(* PLC project TC3_TE1400_GeneratedModule_TctSmplTempCtrl__FB, Beckhoff Automation GmbH & Co. KG TwinCAT 3 Function - TE1400 1.2.1230 *)
(* stored: companyURL www.beckhoff.com, creationDateTime 2018-02-26T08:09:58 *)

TYPE E_TcMatSimDataAreaType : (NotSpecified := 0, Standard, InputSrc, InputDst, OutputSrc, OutputDst, InternalDa, MArea, RetainDa);
END_TYPE

TYPE ST_TcMatSimObjectDataAreaInfo : STRUCT
  pPlcVar : PVOID;
  pModuleProcImg : PVOID;
  nSize : UDINT;
  nDataAreaId : UDINT;
  eDataAreaType : E_TcMatSimDataAreaType;
END_STRUCT;
END_TYPE

{attribute 'pack_mode' := '4'}
TYPE ST_TctSmplTempCtrl_InitData : STRUCT
  Header : TComInitDataHdr;
  CallByHdr : TComInitDataElmHdr;
  CallBy : TctModuleCallByType;
  ExecutionSequenceHdr : TComInitDataElmHdr;
  ExecutionSequence : TctModuleExecutionSequenceType;
  StepSizeHdr : TComInitDataElmHdr;
  StepSize : TctStepSizeType;
  ExtModeParametersHdr : TComInitDataElmHdr;
  ExtModeParameters : TctExtModeParametersType;
  ExecuteModelCodeHdr : TComInitDataElmHdr;
  ExecuteModelCode : BOOL;
  ModelParametersHdr : TComInitDataElmHdr;
  ModelParameters : P_TctSmplTempCtrl_T;
  ContextInfoArr_0_TaskOidHdr : TComInitDataElmHdr;
  ContextInfoArr_0_TaskOid : OTCID;
  ContextInfoArr_0_TaskPriorityHdr : TComInitDataElmHdr;
  ContextInfoArr_0_TaskPriority : UDINT;
  ContextInfoArr_0_TaskCycleTimeNsHdr : TComInitDataElmHdr;
  ContextInfoArr_0_TaskCycleTimeNs : UDINT;
  ContextInfoArr_0_TaskPortHdr : TComInitDataElmHdr;
  ContextInfoArr_0_TaskPort : UINT;
  ContextInfoArr_0_TaskSortOrderHdr : TComInitDataElmHdr;
  ContextInfoArr_0_TaskSortOrder : UDINT;
END_STRUCT;
END_TYPE

TYPE ST_TctSmplTempCtrl_Input : STRUCT
  FeedbackTemp : INT;
END_STRUCT;
END_TYPE

TYPE ST_TctSmplTempCtrl_Output : STRUCT
  HeaterOn : BOOL;
  MonitoringSignals : MonitoringSignalsType;
END_STRUCT;
END_TYPE

FUNCTION_BLOCK FB_TcMatSimObject
  VAR_INPUT
    bWriteFbInputValues : BOOL := TRUE;  (* set this flag to write FB input values to the TcComObject's input DataAreas. This will overwrite the mapped input values before module execution. Set to FALSE to read the mapped input values from the TcComObject to the FB. *)
  END_VAR
  VAR
    pDataAreas : POINTER TO ST_TcMatSimObjectDataAreaInfo;  (* process image src and dst pointers and sizes *)
    nDataAreas : UDINT;
    ipObjSrv : ITComObjectServer;  (* global interface pointers *)
    ipTcComObj : ITComObject;  (* object interface pointers *)
    ipTcCyclic : ITcCyclic;
    ipTcPostCyclic : ITcPostCyclic;
    ipTcAdi : ITcADI;
    ipTask : ITcTask;  (* task interface pointers *)
    pInitData : POINTER TO TComInitDataHdr;  (* initial parameters *)
    hResult : HRESULT;  (* hResult of interface calls (0 if no error) *)
    moduleClsId : CLSID;  (* module class ID *)
    assignedClsId : CLSID;  (* expected/desired module class ID *)
    bClassIdVerified : BOOL;
    bDynInstance : BOOL;  (* flag indicating whether the module instance was created dynamically *)
    eInitialObjState : TCOM_STATE := TCOM_STATE.TCOM_STATE_INIT;  (* the object state at the time FB_init was called, FB_exit will try to switch to this state (only if this means to shift down) *)
  END_VAR

            
          

{attribute 'object_name' := 'ReleaseTcComInterface'}
METHOD ReleaseTcComInterface : HRESULT
  VAR
    nStateChangeCnt : DINT := 0;
  END_VAR
                  
IF (ipTcComObj<>0) THEN
  WHILE (State>eInitialObjState AND nStateChangeCnt<1000) DO
    State := eInitialObjState;
    nStateChangeCnt := nStateChangeCnt+1;
  END_WHILE
  ReleaseObjInterfaces();
  IF (bDynInstance) THEN
    ReleaseTcComInterface := TC3_MODULE.FW_ObjMgr_DeleteInstance(ADR(ipTcComObj));
  ELSE
    ipTcComObj.TcRelease();
  END_IF
  ipTcComObj := 0;
END_IF
                  
                
END_METHOD

{attribute 'object_name' := 'ReleaseObjInterfaces'}
METHOD ReleaseObjInterfaces : HRESULT
                  
// release interface pointers
IF (ipTcCyclic<>0) THEN
  ipTcCyclic.TcRelease();
  ipTcCyclic := 0;
END_IF
IF (ipTcPostCyclic<>0) THEN
  ipTcPostCyclic.TcRelease();
  ipTcPostCyclic := 0;
END_IF
IF (ipTcAdi<>0) THEN
  ipTcAdi.TcRelease();
  ipTcAdi := 0;
END_IF
                  
                
END_METHOD

{attribute 'object_name' := 'Internal_SetObjState'}
METHOD Internal_SetObjState
  VAR_INPUT
    hr : REFERENCE TO HRESULT;
    nextState : TCOM_STATE;
  END_VAR
                  
// verify class id
IF (SUCCEEDED(hr)) THEN
  hr := VerifyClassId();
END_IF

// switch object state
IF (SUCCEEDED(hr) AND nextState>=TCOM_STATE_INIT) THEN
  IF (ipTcComObj=0) THEN
    hr := Tc2_System.E_HRESULTAdsErr.NOINTERFACE;
  END_IF
  IF (ipObjSrv=0) THEN
    hr := Tc2_System.E_HRESULTAdsErr.NOINTERFACE;
  END_IF
  IF (SUCCEEDED(hr)) THEN
    hr := ipTcComObj.TcSetObjState(nextState,ipObjSrv,pInitData);
  END_IF
END_IF
                  
                
END_METHOD

{attribute 'object_name' := 'FB_init'}
METHOD FB_init : BOOL
  VAR_INPUT
    bInitRetains : BOOL;  (* init retain variables *)
    bInCopyCode : BOOL;  (* Online Change *)
    oid : OTCID;
  END_VAR
                  
FB_init := SUCCEEDED(Init(oid));
                  
                
END_METHOD

{attribute 'object_name' := 'GetObjPara'}
METHOD GetObjPara : HRESULT
  VAR_INPUT
    pid : PTCID;
    nData : UDINT;
    pData : PVOID;
  END_VAR
                  
IF (ipTcComObj=0) THEN
  GetObjPara := Tc2_System.E_HRESULTAdsErr.NOINTERFACE;
END_IF

IF (SUCCEEDED(GetObjPara)) THEN
  GetObjPara := ipTcComObj.TcGetObjPara(pid:=pid,nData,pData,0);
END_IF
                  
                
END_METHOD

{attribute 'object_name' := 'QueryObjInterface'}
METHOD QueryObjInterface
  VAR_INPUT
    hr : REFERENCE TO HRESULT;
    iid : REFERENCE TO IID;
    pipItf : POINTER TO ITcUnknown;
  END_VAR
  VAR CONSTANT
    pNull : PVOID := 0;
  END_VAR
                  
IF (SUCCEEDED(hr)) THEN
  IF (ipTcComObj=0) THEN
    hr := Tc2_System.E_HRESULTAdsErr.NOINTERFACE;
  ELSIF (pipItf^=ULINT_TO_DWORD(pNull)) THEN
    hr := ipTcComObj.TcQueryInterface(iid:= iid, pipItf:=pipItf);
  END_IF
END_IF
                  
                
END_METHOD

{attribute 'object_name' := 'SaveOnlineParametersForInit'}
METHOD SaveOnlineParametersForInit : HRESULT
  VAR
    idx : UINT;
    pInitElemHdr : POINTER TO TComInitDataElmHdr;
    pData : PVOID;
    nData : UDINT;
  END_VAR
  VAR CONSTANT
    nInitDataAlignment : UDINT := 4;
  END_VAR
                  IF (pInitData<>0) THEN
  pInitElemHdr := pInitData + SIZEOF(pInitData^);
  FOR idx:=1 TO pInitData^.uiElmCnt DO
    pData := pInitElemHdr + ULINT_TO_DWORD(SIZEOF(pInitElemHdr^));
    nData := pInitElemHdr^.cbData;
    SaveOnlineParametersForInit := GetObjPara(pInitElemHdr^.indexOffset,nData,pData);
    IF (FAILED(SaveOnlineParametersForInit)) THEN
      RETURN;
    END_IF
    pInitElemHdr := pData + (nInitDataAlignment*((nData + nInitDataAlignment - 1)/nInitDataAlignment));
  END_FOR
ELSE
	SaveOnlineParametersForInit := Tc2_System.E_HRESULTAdsErr.NOTINIT;
END_IF
                  
                
END_METHOD

{attribute 'object_name' := 'ResetHresult'}
METHOD ResetHresult
                  hResult := S_OK;
                
END_METHOD

{attribute 'object_name' := 'Execute'}
METHOD Execute : HRESULT
  VAR
    nDaIdx : UDINT;
    pCurDataArea : POINTER TO ST_TcMatSimObjectDataAreaInfo;
  END_VAR
                  
IF (SUCCEEDED(hResult)) THEN
  hResult := VerifyClassId();
END_IF

IF (SUCCEEDED(hResult) AND State<>TCOM_STATE_OP) THEN
  hResult := Tc2_System.E_HRESULTAdsErr.NOTREADY;
END_IF

// get image pointers
IF (SUCCEEDED(hResult)) THEN
  GetImagePtrs(hResult);
END_IF

// copy inputs
IF (pDataAreas<>0 AND nDataAreas>0 AND bWriteFbInputValues) THEN
  FOR nDaIdx:=0 TO nDataAreas-1 DO
    IF (FAILED(hResult))THEN
      CONTINUE;
    END_IF
    pCurDataArea := pDataAreas + nDaIdx*SIZEOF(ST_TcMatSimObjectDataAreaInfo);
    IF ((pCurDataArea^.eDataAreaType <> E_TcMatSimDataAreaType.InputDst))THEN
      CONTINUE;
    END_IF
    IF (pCurDataArea^.pModuleProcImg<>0 AND pCurDataArea^.pPlcVar<>0) THEN
      MEMCPY(pCurDataArea^.pModuleProcImg,pCurDataArea^.pPlcVar,pCurDataArea^.nSize);
    ELSE
      hResult := Tc2_System.E_HRESULTAdsErr.NOINTERFACE;
    END_IF
  END_FOR
END_IF

// call cycle update
IF (SUCCEEDED(hResult)) THEN
  IF (ipTcCyclic<>0) THEN
    hResult := ipTcCyclic.CycleUpdate(ipTask:= ipTask, ipCaller:= 0, context:= 0);
  ELSE
    hResult := Tc2_System.E_HRESULTAdsErr.NOINTERFACE;
  END_IF
END_IF

// copy outputs
IF (pDataAreas<>0 AND nDataAreas>0) THEN
  FOR nDaIdx:=0 TO nDataAreas-1 DO
    IF (FAILED(hResult))THEN
      CONTINUE;
    END_IF
    pCurDataArea := pDataAreas + nDaIdx*SIZEOF(ST_TcMatSimObjectDataAreaInfo);
    IF ((pCurDataArea^.eDataAreaType = E_TcMatSimDataAreaType.OutputSrc) OR NOT bWriteFbInputValues) THEN
      IF (pCurDataArea^.pModuleProcImg<>0 AND pCurDataArea^.pPlcVar<>0) THEN
        MEMCPY(pCurDataArea^.pPlcVar,pCurDataArea^.pModuleProcImg,pCurDataArea^.nSize);
      ELSE
        hResult := Tc2_System.E_HRESULTAdsErr.NOINTERFACE;
      END_IF
    END_IF
  END_FOR
END_IF


// call post cyclic update
IF (SUCCEEDED(hResult)) THEN
  IF (ipTcPostCyclic<>0) THEN
    hResult := ipTcPostCyclic.PostCyclicUpdate(ipTask:= 0, ipCaller:= 0, context:= 0);
  ELSE
    hResult := Tc2_System.E_HRESULTAdsErr.NOINTERFACE;
  END_IF
END_IF

ReleaseImagePtrs();

Execute := hResult;
                  
                
END_METHOD

{attribute 'object_name' := 'GetImagePtrs'}
METHOD GetImagePtrs
  VAR_INPUT
    hr : REFERENCE TO HRESULT;
  END_VAR
  VAR
    nDaIdx : UDINT;
    pCurDataArea : POINTER TO ST_TcMatSimObjectDataAreaInfo;
  END_VAR
                  
IF (ipTcAdi=0) THEN
  hr := Tc2_System.E_HRESULTAdsErr.NOINTERFACE;
END_IF
IF(State<>TCOM_STATE_OP)THEN
  hr := Tc2_System.E_HRESULTAdsErr.INVALIDSTATE;
END_IF


// get pointers to process images
IF (pDataAreas<>0 AND nDataAreas>0) THEN
  FOR nDaIdx:=0 TO nDataAreas-1 DO
    pCurDataArea := pDataAreas + nDaIdx*SIZEOF(ST_TcMatSimObjectDataAreaInfo);
    IF (FAILED(hr))THEN
      CONTINUE;
    END_IF
    IF ((pCurDataArea^.eDataAreaType <> E_TcMatSimDataAreaType.InputDst) AND (pCurDataArea^.eDataAreaType <> E_TcMatSimDataAreaType.OutputSrc))THEN
      CONTINUE;
    END_IF
    IF (pCurDataArea^.pModuleProcImg=0 AND pCurDataArea^.nSize>0) THEN
      hr := ipTcAdi.GetImagePtr(size:= pCurDataArea^.nSize , offs:=0 , adi_x:=pCurDataArea^.nDataAreaId , ppData:=ADR(pCurDataArea^.pModuleProcImg));
    END_IF
  END_FOR
END_IF

IF (FAILED(hr)) THEN
  ReleaseImagePtrs();
END_IF
                  
                
END_METHOD

{attribute 'object_name' := 'VerifyClassId'}
METHOD VerifyClassId : HRESULT
  VAR
    emptyClsId : CLSID;
  END_VAR
                  memset(ADR(emptyClsId),0,SIZEOF(emptyClsId));
IF (bClassIdVerified) THEN
  // class ID was already verified
  VerifyClassId := Tc2_System.E_HRESULTAdsErr.HRESULT_ADS_NOERROR;
ELSIF (memcmp(ADR(assignedClsId),ADR(emptyClsId),SIZEOF(assignedClsId))=0) THEN
  // skip class ID verification if no assignedClsId specified
  VerifyClassId := Tc2_System.E_HRESULTAdsErr.HRESULT_ADS_NOERROR;
ELSE
  // verify class ID
  VerifyClassId := ReadModuleClassId();

  IF (SUCCEEDED(VerifyClassId)) THEN
    IF (memcmp(ADR(assignedClsId),ADR(moduleClsId),SIZEOF(assignedClsId))<>0) THEN
     VerifyClassId := Tc2_System.E_HRESULTAdsErr.INVALIDCLSID;
    END_IF
  END_IF
  bClassIdVerified := SUCCEEDED(VerifyClassId);
END_IF
                  
                
END_METHOD

{attribute 'object_name' := 'SetObjPara'}
METHOD SetObjPara : HRESULT
  VAR_INPUT
    pid : PTCID;
    nData : UDINT;
    pData : PVOID;
  END_VAR
                  
IF (ipTcComObj=0) THEN
  SetObjPara := Tc2_System.E_HRESULTAdsErr.NOINTERFACE;
END_IF

IF (SUCCEEDED(SetObjPara)) THEN
  SetObjPara := ipTcComObj.TcSetObjPara(pid:=pid,nData,pData,0);
END_IF
                  
                
END_METHOD

{attribute 'object_name' := 'QueryTcComInterface'}
METHOD QueryTcComInterface
  VAR_INPUT
    hr : REFERENCE TO HRESULT;
    oid : OTCID;
  END_VAR
                  
IF (ipObjSrv=0) THEN
  hr := Tc2_System.E_HRESULTAdsErr.NOINTERFACE;
END_IF

IF (SUCCEEDED(hr) AND ipTcComObj=0) THEN
  bDynInstance := FALSE;
  IF(oid>0) THEN
    // query interface of existing object
    hr := ipObjSrv.TcQueryObjectInterface(oid,IID_ITComObject,ADR(ipTcComObj));
  ELSE
    // create new instance and get the object interface
    hr := ipObjSrv.TcCreateInstance(assignedClsId,IID_ITComObject,ADR(ipTcComObj));
    IF (SUCCEEDED(hr)) THEN
      bDynInstance := TRUE;
      hr := ipTcComObj.TcSetObjectId(OTCID_CreateNewId);
    END_IF
  END_IF
  IF (SUCCEEDED(hr)) THEN
    eInitialObjState := State;
  END_IF
END_IF
                  
                
END_METHOD

{attribute 'object_name' := 'ReleaseImagePtrs'}
METHOD ReleaseImagePtrs : HRESULT
  VAR
    nDaIdx : UDINT;
    pCurDataArea : POINTER TO ST_TcMatSimObjectDataAreaInfo;
  END_VAR
                  
IF (ipTcAdi=0) THEN
  ReleaseImagePtrs := Tc2_System.E_HRESULTAdsErr.NOINTERFACE;
END_IF

IF (SUCCEEDED(ReleaseImagePtrs) AND pDataAreas<>0 AND nDataAreas>0) THEN
  // release pointers to the simulink module process images
  FOR nDaIdx:=0 TO nDataAreas-1 DO
    pCurDataArea := pDataAreas + nDaIdx*SIZEOF(ST_TcMatSimObjectDataAreaInfo);

    IF (pCurDataArea^.pModuleProcImg<>0) THEN
      ipTcAdi.ReleaseImagePtr(pData:=pCurDataArea^.pModuleProcImg);
      pCurDataArea^.pModuleProcImg := 0;
    END_IF
  END_FOR
END_IF
                  
                
END_METHOD

{attribute 'object_name' := 'FB_exit'}
METHOD FB_exit : BOOL
  VAR_INPUT
    bInCopyCode : BOOL;  (* Online Change *)
  END_VAR
                  
IF (NOT bInCopyCode) THEN
  IF (ipObjSrv<>0) THEN
    ipObjSrv.TcRelease();
    ipObjSrv := 0;
  END_IF

  ReleaseTcComInterface();
END_IF
                  
                
END_METHOD

{attribute 'object_name' := 'InitObjName'}
METHOD InitObjName
  VAR_INPUT
    hr : REFERENCE TO HRESULT;
  END_VAR
  VAR
    objectName : STRING(255) := 'TcMatSimObject_PlcRtFbInstance';
    oid : OTCID;
  END_VAR
                  
IF (SUCCEEDED(hr)) THEN
  hr := ipTcComObj.TcGetObjectId(oid);
END_IF

IF (SUCCEEDED(hr) and bDynInstance) THEN
  objectName := TC2_STANDARD.CONCAT(objectName,'_');
  objectName := TC2_STANDARD.CONCAT(objectName,UDINT_TO_STRING(oid));
  hr := ipTcComObj.TcSetObjectName(ADR(objectName));
END_IF
                  
                
END_METHOD

{attribute 'object_name' := 'SetObjState'}
METHOD SetObjState : HRESULT
  VAR_INPUT
    finalState : TCOM_STATE;
  END_VAR
  VAR
    bShiftUp : BOOL;
    bShiftDown : BOOL;
    currentState : TCOM_STATE;
  END_VAR
                  
currentState := State;

bShiftUp := finalState>currentState;
bShiftDown := finalState<currentState;

// do not switch up on error
IF (FAILED(hresult)) THEN
  bShiftUp := FALSE;
END_IF
// reset existing error on switching down
IF (bShiftDown) THEN
  ResetHresult();
END_IF

// prepared state switch
CASE currentState OF
  TCOM_STATE_INIT:
    IF(bShiftUp) THEN
      QueryTcComInterface(hResult,0);
      Internal_SetObjState(hResult,TCOM_STATE.TCOM_STATE_PREOP);
      InitObjName(hResult);
    END_IF

  TCOM_STATE_PREOP:
    IF(bShiftUp) THEN
      Internal_SetObjState(hResult,TCOM_STATE.TCOM_STATE_SAFEOP);
      QueryObjInterfaces(hResult);
    ELSIF (bShiftDown) THEN
      Internal_SetObjState(hResult,TCOM_STATE.TCOM_STATE_INIT);
    END_IF

  TCOM_STATE_SAFEOP:
    IF(bShiftUp) THEN
      Internal_SetObjState(hResult,TCOM_STATE.TCOM_STATE_OP);
      QueryObjInterfaces(hResult);
    ELSIF (bShiftDown) THEN
      Internal_SetObjState(hResult,TCOM_STATE.TCOM_STATE_PREOP);
      ReleaseObjInterfaces();
    END_IF


  TCOM_STATE_OP:
    IF (bShiftDown) THEN
      Internal_SetObjState(hResult,TCOM_STATE.TCOM_STATE_SAFEOP);
    END_IF
END_CASE

SetObjState := hResult;
                  
                
END_METHOD

{attribute 'object_name' := 'QueryObjInterfaces'}
METHOD QueryObjInterfaces
  VAR_INPUT
    hr : REFERENCE TO HRESULT;
  END_VAR
                  
IF(State<TCOM_STATE_PREOP)THEN
  hr := Tc2_System.E_HRESULTAdsErr.INVALIDSTATE;
END_IF

//cyclic interface
QueryObjInterface(hr,IID_ITCCYCLIC,ADR(ipTcCyclic));
//post cyclic interface
QueryObjInterface(hr,IID_ITCPOSTCYCLIC,ADR(ipTcPostCyclic));
//adi interface
QueryObjInterface(hr,IID_ITcADI,ADR(ipTcAdi));
                  
                
END_METHOD

{attribute 'object_name' := 'Init'}
METHOD Init : HRESULT
  VAR_INPUT
    oid : OTCID;
  END_VAR
                  
// preinitialize variables
memset(ADR(moduleClsId),0,SIZEOF(moduleClsId));
bClassIdVerified := FALSE;
hResult := Tc2_System.E_HRESULTAdsErr.HRESULT_ADS_NOERROR;

// get object server
IF (ipObjSrv=0) THEN
  hResult := FW_ObjMgr_GetObjectServer(_AppInfo.ObjId,ADR(ipObjSrv));
END_IF

// try to get object interfaces
IF (SUCCEEDED(hresult)) THEN
  QueryTcComInterface(hResult,oid);
END_IF

// verify class id
IF (SUCCEEDED(hresult)) THEN
  hresult := VerifyClassId();
END_IF

// query interfaces, if the current state is higher than INIT
IF (SUCCEEDED(hresult) AND State>TCOM_STATE.TCOM_STATE_INIT) THEN
  QueryObjInterfaces(hResult);
END_IF

// return value
Init := hresult;
                  
                
END_METHOD

{attribute 'object_name' := 'ReadModuleClassId'}
METHOD ReadModuleClassId : HRESULT
  VAR
    emptyClsId : CLSID;
  END_VAR
                  memset(ADR(emptyClsId),0,SIZEOF(emptyClsId));
IF (memcmp(ADR(moduleClsId),ADR(emptyClsId),SIZEOF(moduleClsId))=0) THEN
  IF (ipTcComObj=0) THEN
    ReadModuleClassId := Tc2_System.E_HRESULTAdsErr.NOINTERFACE;
  END_IF

  //objectClsId := clsid;
  IF (SUCCEEDED(ReadModuleClassId)) THEN
    ReadModuleClassId := ipTcComObj.GetClassId(moduleClsId);
  END_IF
END_IF
                
END_METHOD

METHOD PUBLIC AssignClassId
VAR_INPUT
	clsId : CLSID;
END_VAR
                  assignedClsId := clsId;
bClassIdVerified := false;
                  
                
END_METHOD

PROPERTY Error : BOOL
GET
                    Error := FAILED(hResult);
                  
END_GET
END_PROPERTY

METHOD PUBLIC SetDataAreaInfo
VAR_INPUT
  pDataAreas: POINTER TO ST_TcMatSimObjectDataAreaInfo;
  nDataAreas: UDINT;
END_VAR
                  
THIS^.nDataAreas := nDataAreas;
THIS^.pDataAreas := pDataAreas;
                  
                
END_METHOD

METHOD PUBLIC SetInitDataInfo
VAR_INPUT
  pInitData : POINTER TO TComInitDataHdr;
END_VAR
                  this^.pInitData := pInitData;
                
END_METHOD

PROPERTY ClassId : CLSID
GET
                    hResult := ReadModuleClassId();
ClassId := moduleClsId;
                    
                  
END_GET
END_PROPERTY

PROPERTY State : TCOM_STATE
GET
  VAR
    hr : HRESULT := S_OK;
    eObjState : TCOM_STATE;
  END_VAR
                    
IF (ipTcComObj<>0) THEN
  hr := ipTcComObj.TcGetObjState(ADR(eObjState));
IF (FAILED(hr)) THEN
  eObjState := TCOM_STATE.TCOM_STATE_INIT;
END_IF
ELSE
  eObjState := TCOM_STATE.TCOM_STATE_INIT;
END_IF
State := eObjState;
                    
                  
END_GET
SET
                    SetObjState(State);
                  
END_SET
END_PROPERTY

PROPERTY ErrorCode : HRESULT
GET
                    ErrorCode := hResult;
                  
END_GET
END_PROPERTY
END_FUNCTION_BLOCK

{attribute 'TcDependOnClassFactory' := 'TctSmplTempCtrl_'}
FUNCTION_BLOCK FB_TctSmplTempCtrl_ EXTENDS FB_TcMatSimObject
  VAR_INPUT
    stInput : ST_TctSmplTempCtrl_Input;
  END_VAR
  VAR_OUTPUT
    stOutput : ST_TctSmplTempCtrl_Output;
  END_VAR
  VAR
    stInitData : ST_TctSmplTempCtrl_InitData;
    arrDataAreas : ARRAY[1..2] OF ST_TcMatSimObjectDataAreaInfo;
    bParametersVerified : BOOL;
  END_VAR

            
          

{attribute 'object_name' := 'Internal_SetObjState'}
METHOD Internal_SetObjState
  VAR_INPUT
    hr : REFERENCE TO HRESULT;
    nextState : TCOM_STATE;
  END_VAR
                  
// update pointer to InitData structure
SetInitDataInfo(ADR(stInitData));
// call base method
SUPER^.Internal_SetObjState(hr,nextState);
                  
                
END_METHOD

{attribute 'object_name' := 'SaveOnlineParametersForInit'}
METHOD SaveOnlineParametersForInit : HRESULT
  VAR
    idx : UINT;
    pInitElemHdr : POINTER TO TComInitDataElmHdr;
    pData : PVOID;
    nData : UDINT;
  END_VAR
  VAR CONSTANT
    nInitDataAlignment : UDINT := 4;
  END_VAR
                  
// update pointer to InitData structure
SetInitDataInfo(ADR(stInitData));
// call base method
SaveOnlineParametersForInit := SUPER^.SaveOnlineParametersForInit();
                  
                
END_METHOD

METHOD FB_init : BOOL
  VAR_INPUT
    bInitRetains : BOOL;  (* if TRUE, the retain variables are initialized (warm start / cold start) *)
    bInCopyCode : BOOL;  (* if TRUE, the instance afterwards gets moved into the copy code (online change) *)
    oid : OTCID;
  END_VAR
  VAR
    clsId : CLSID;
  END_VAR
                  
// initialize flags
bParametersVerified := false;
                    
// set module class id for compatibility check
clsId.Data1 := 16#0b213a0b;
clsId.Data2 := 16#44ab;
clsId.Data3 := 16#4974;
clsId.Data4[0] := 16#90;
clsId.Data4[1] := 16#46;
clsId.Data4[2] := 16#05;
clsId.Data4[3] := 16#c8;
clsId.Data4[4] := 16#6a;
clsId.Data4[5] := 16#96;
clsId.Data4[6] := 16#15;
clsId.Data4[7] := 16#97;

AssignClassId(clsId);
                    
// initialize InitData structure with default values              
stInitData.CallByHdr.indexGroup := 0;
stInitData.CallByHdr.indexOffset := 16#00000000;
stInitData.CallByHdr.cbData := SIZEOF(stInitData.CallBy);
stInitData.CallBy := TctModuleCallByType.CyclicTask;
stInitData.ExecutionSequenceHdr.indexGroup := 0;
stInitData.ExecutionSequenceHdr.indexOffset := 16#00000001;
stInitData.ExecutionSequenceHdr.cbData := SIZEOF(stInitData.ExecutionSequence);
stInitData.ExecutionSequence := TctModuleExecutionSequenceType.StateUpdateAfterOutputMapping;
stInitData.StepSizeHdr.indexGroup := 0;
stInitData.StepSizeHdr.indexOffset := 16#00000002;
stInitData.StepSizeHdr.cbData := SIZEOF(stInitData.StepSize);
stInitData.StepSize := TctStepSizeType.RequireMatchingTaskCycleTime;
stInitData.ExtModeParametersHdr.indexGroup := 0;
stInitData.ExtModeParametersHdr.indexOffset := 16#bf002000;
stInitData.ExtModeParametersHdr.cbData := SIZEOF(stInitData.ExtModeParameters);
stInitData.ExtModeParameters.ConnectionTimeout := 3;
stInitData.ExtModeParameters.InitIncomingPktBufferSize := 10000;
stInitData.ExtModeParameters.InitOutgoingPktBufferSize := 10000;
stInitData.ExtModeParameters.Activated := 1;
stInitData.ExtModeParameters.AllowExecutionCommands := 0;
stInitData.ExtModeParameters.WaitForStartCommand := 0;
stInitData.ExtModeParameters.AllowParameterChange := 0;
stInitData.ExecuteModelCodeHdr.indexGroup := 0;
stInitData.ExecuteModelCodeHdr.indexOffset := 16#00000007;
stInitData.ExecuteModelCodeHdr.cbData := SIZEOF(stInitData.ExecuteModelCode);
stInitData.ExecuteModelCode := 1;
stInitData.ModelParametersHdr.indexGroup := 0;
stInitData.ModelParametersHdr.indexOffset := 16#83000000;
stInitData.ModelParametersHdr.cbData := SIZEOF(stInitData.ModelParameters);
stInitData.ModelParameters.Kp := 50;
stInitData.ModelParameters.Tn := 200;
stInitData.ModelParameters.sawtooth_rep_seq_y[0] := 0;
stInitData.ModelParameters.sawtooth_rep_seq_y[1] := 60;
stInitData.ModelParameters.PI_y_max := 60;
stInitData.ModelParameters.PI_y_min := 0;
stInitData.ModelParameters.InternalSetpoint_Value := 37;
stInitData.ModelParameters.scale_Gain := 0.1;
stInitData.ModelParameters.Integrator_IC := 0;
stInitData.ModelParameters.Constant_Value := 0.1;
stInitData.ModelParameters.LookUpTable1_bp01Data[0] := 0;
stInitData.ModelParameters.LookUpTable1_bp01Data[1] := 0.1;
stInitData.ContextInfoArr_0_TaskOidHdr.indexGroup := 0;
stInitData.ContextInfoArr_0_TaskOidHdr.indexOffset := 16#03002060;
stInitData.ContextInfoArr_0_TaskOidHdr.cbData := SIZEOF(stInitData.ContextInfoArr_0_TaskOid);
stInitData.ContextInfoArr_0_TaskPriorityHdr.indexGroup := 0;
stInitData.ContextInfoArr_0_TaskPriorityHdr.indexOffset := 16#03002070;
stInitData.ContextInfoArr_0_TaskPriorityHdr.cbData := SIZEOF(stInitData.ContextInfoArr_0_TaskPriority);
stInitData.ContextInfoArr_0_TaskCycleTimeNsHdr.indexGroup := 0;
stInitData.ContextInfoArr_0_TaskCycleTimeNsHdr.indexOffset := 16#03002080;
stInitData.ContextInfoArr_0_TaskCycleTimeNsHdr.cbData := SIZEOF(stInitData.ContextInfoArr_0_TaskCycleTimeNs);
stInitData.ContextInfoArr_0_TaskPortHdr.indexGroup := 0;
stInitData.ContextInfoArr_0_TaskPortHdr.indexOffset := 16#03002090;
stInitData.ContextInfoArr_0_TaskPortHdr.cbData := SIZEOF(stInitData.ContextInfoArr_0_TaskPort);
stInitData.ContextInfoArr_0_TaskSortOrderHdr.indexGroup := 0;
stInitData.ContextInfoArr_0_TaskSortOrderHdr.indexOffset := 16#030020b0;
stInitData.ContextInfoArr_0_TaskSortOrderHdr.cbData := SIZEOF(stInitData.ContextInfoArr_0_TaskSortOrder);
stInitData.Header.cbData := SIZEOF(stInitData)-SIZEOF(stInitData.Header);
stInitData.Header.uiElmCnt := 11;


// set pointer to InitData structure
SetInitDataInfo(ADR(stInitData));

// set DataArea information
SetDataAreaInfo(ADR(arrDataAreas),2);
arrDataAreas[1].nDataAreaId := 0;
arrDataAreas[1].nSize := SIZEOF(stInput);
arrDataAreas[1].pPlcVar := ADR(stInput);
arrDataAreas[1].pModuleProcImg := 0;
arrDataAreas[1].eDataAreaType := E_TcMatSimDataAreaType.InputDst;
arrDataAreas[2].nDataAreaId := 1;
arrDataAreas[2].nSize := SIZEOF(stOutput);
arrDataAreas[2].pPlcVar := ADR(stOutput);
arrDataAreas[2].pModuleProcImg := 0;
arrDataAreas[2].eDataAreaType := E_TcMatSimDataAreaType.OutputSrc;


// initialize basic interface pointers and return
FB_init := SUCCEEDED(Init(oid));
                  
                
END_METHOD

METHOD Execute : HRESULT
                  
IF (SUCCEEDED(hResult)) THEN
  hResult := VerifyParameters();
END_IF

// update DataArea information
SetDataAreaInfo(ADR(arrDataAreas),2);
arrDataAreas[1].nDataAreaId := 0;
arrDataAreas[1].nSize := SIZEOF(stInput);
arrDataAreas[1].pPlcVar := ADR(stInput);
arrDataAreas[1].pModuleProcImg := 0;
arrDataAreas[1].eDataAreaType := E_TcMatSimDataAreaType.InputDst;
arrDataAreas[2].nDataAreaId := 1;
arrDataAreas[2].nSize := SIZEOF(stOutput);
arrDataAreas[2].pPlcVar := ADR(stOutput);
arrDataAreas[2].pModuleProcImg := 0;
arrDataAreas[2].eDataAreaType := E_TcMatSimDataAreaType.OutputSrc;

	
// call base method
Execute := SUPER^.Execute();
                  
                
END_METHOD

{attribute 'object_name' := 'VerifyParameters'}
METHOD VerifyParameters : HRESULT
  VAR
    moduleCallByParam : TctModuleCallByType;
  END_VAR
                  
IF (bParametersVerified) THEN
  VerifyParameters := Tc2_System.E_HRESULTAdsErr.HRESULT_ADS_NOERROR;
ELSE
  VerifyParameters := GetObjPara(stInitData.CallByHdr.indexOffset,SIZEOF(moduleCallByParam),ADR(moduleCallByParam));
  
  // check the "CallBy" parameter to be set to "Module"
  IF (SUCCEEDED(VerifyParameters) AND (moduleCallByParam <> TctModuleCallByType.Module)) THEN
      VerifyParameters := Tc2_System.E_HRESULTAdsErr.INVALIDPARM;
  END_IF
  
  // set the parameters verified flag
  bParametersVerified := SUCCEEDED(VerifyParameters);
END_IF
                  
                
END_METHOD

PROPERTY InitData : ST_TctSmplTempCtrl_InitData
GET
                    InitData := stInitData;
                  
END_GET
SET
                    stInitData := InitData;
                  
END_SET
END_PROPERTY
END_FUNCTION_BLOCK
